{attribute 'qualified_only'}
{attribute 'strict'}
TYPE E_InverterError :
(
	nOF := 0,
	InF := 1,
	CFF := 3,
	CFI := 4,
	SLF1:= 5, 
	EPF1:= 8,
	OCF := 9,
	CrF1:= 10,
	OHF := 16,
	OLF := 17,
	ObF := 18,
	OSF := 19,
	OPF1:= 20,
	PHF := 21,
	USF := 22,
	SCF1:= 23,
	SOF := 24,
	tnF := 25,
	InF1:= 26,
	InF2:= 27,
	InF3:= 28,
	InF4:= 29,
	SCF3:= 32,
	OPF2:= 33,
	SLF2:= 42,
	SLF3:= 45,
	InF9:= 51,
	InFb:= 53,
	tJF := 54,
	SCF4:= 55,
	SCF5:= 56,
	InFE:= 69, 
	CFI2:= 77,
	ULF := 100,
	OLC := 101,
	SPIF:= 102,
	LFF1:= 106
	
)WORD;
END_TYPE

(* stored: Version 1.1.0.1, ProductVersion 3.1.4024.12
   EnumerationTextList E_InverterError: Id {2e727e13-9486-477d-a6d8-30c64fff4769} *)
